{attribute addProperty BoxType "EJ3318-0000-0017"}
{attribute addProperty Id "TC_ChannelAT %I*ARRAY[0..14] OF TC_Channel_17AE08DB256320RTD_Inputs_ChannelAT %I*ARRAY[0..2] OF RTD_Inputs_Channel_17AE08DB6480WcStateAT %I*WcState_98A4DF7520.250InfoDataAT %I*InfoData_BC63D37F80100"}
{attribute addProperty CRC "604556167"}
{attribute addProperty SizeInBites "402"}
{attribute addProperty SizeInBytes "50.25"}
TYPE EJ3318_4B9E477A :
STRUCT
	{attribute addProperty Name "TC_Channel"}
	TC_Channel : ARRAY[0..14] OF TC_Channel_17AE08DB;
	{attribute addProperty Name "RTD_Inputs_Channel"}
	RTD_Inputs_Channel : ARRAY[0..2] OF RTD_Inputs_Channel_17AE08DB;
	{attribute addProperty Name "WcState"}
	WcState : WcState_98A4DF75;
	{attribute addProperty Name "InfoData"}
	InfoData : InfoData_BC63D37F;
END_STRUCT
END_TYPE

(* stored: Version 1.2.0.0, ProductVersion 3.1.4024.9
   DUT EJ3318_4B9E477A: Id {d5aee36e-8c75-4423-a139-637ea4a5e236} *)
